///EL1088 | 8-channel digital input terminal 24 V DC, 3 ms, negative switching
FUNCTION_BLOCK EL1088_v1_00
VAR_INPUT
	En: BOOL;
END_VAR
VAR_OUTPUT
	EnO: BOOL;
	bDi_1: BOOL;
	bDi_2: BOOL;
	bDi_3: BOOL;
	bDi_4: BOOL;
	bDi_5: BOOL;
	bDi_6: BOOL;
	bDi_7: BOOL;
	bDi_8: BOOL;
	bError: BOOL;
END_VAR
VAR
	Channel_1_Input AT %I*: BOOL;
	Channel_2_Input AT %I*: BOOL;
	Channel_3_Input AT %I*: BOOL;
	Channel_4_Input AT %I*: BOOL;
	Channel_5_Input AT %I*: BOOL;
	Channel_6_Input AT %I*: BOOL;
	Channel_7_Input AT %I*: BOOL;
	Channel_8_Input AT %I*: BOOL;
	WcState_WcState AT %I*: BOOL;
	InfoData_State AT %I*: UINT;
END_VAR

EnO:=En;

IF En AND (WcState_WcState OR InfoData_State<>16#8) THEN
	bError:=TRUE;
ELSE
	bError:=FALSE;
END_IF

IF En THEN
	IF bError=FALSE THEN
		bDi_1:=Channel_1_Input;
		bDi_2:=Channel_2_Input;
		bDi_3:=Channel_3_Input;
		bDi_4:=Channel_4_Input;
		bDi_5:=Channel_5_Input;
		bDi_6:=Channel_6_Input;
		bDi_7:=Channel_7_Input;
		bDi_8:=Channel_8_Input;
	ELSE
		bDi_1:=FALSE;
		bDi_2:=FALSE;
		bDi_3:=FALSE;
		bDi_4:=FALSE;
		bDi_5:=FALSE;
		bDi_6:=FALSE;
		bDi_7:=FALSE;
		bDi_8:=FALSE;
	END_IF
END_IF

END_FUNCTION_BLOCK

(* stored: Version 1.1.0.1, ProductVersion 3.1.0.25
   POU EL1088_v1_00: Id {283a2226-cbff-4e8a-a59b-5b160e75d786} *)
